PROGRAM MAIN
VAR
	fb_statemachine : FB_StateMachine;
END_VAR

fb_statemachine();

END_PROGRAM

(* stored: Version 1.1.0.1, ProductVersion 3.1.4024.13
   POU MAIN: Id {6dd6ae82-dd44-4e79-8cfe-c1b243a8067c}, SpecialFunc None *)
